{attribute 'linkalways'} 
{attribute 'no_explicit_call' := 'This FB is a CLASS and must be accessed using methods or properties'}
{attribute 'enable_dynamic_creation'}
FUNCTION_BLOCK Node_FB_VN_InitializeFunction EXTENDS VisionNode
VAR
    eFunction : _ETcVnInitializableFunction(ETcVnInitializableFunction.TCVN_IF_OCR);
    nOptions : _ULINT(0);
    bStart : _BOOL(FALSE);
    //nTimeout : 
	hresult : _HRESULT(S_OK);
END_VAR

// This is currently disabled as it's an FB and not a function.

METHOD PUBLIC  Clone : I_Node
VAR
	pNode : POINTER TO Node_FB_VN_InitializeFunction;
END_VAR
pNode := __NEW(Node_FB_VN_InitializeFunction);
Clone := pNode^;
END_METHOD

METHOD FB_init : BOOL
VAR_INPUT
	bInitRetains : BOOL; // if TRUE, the retain variables are initialized (warm start / cold start)
	bInCopyCode : BOOL;  // if TRUE, the instance afterwards gets moved into the copy code (online change)
END_VAR
AddParameter('eFunction', eFunction);
AddParameter('nOptions', nOptions);
AddParameter('bStart', bStart);
//AddParameter('nTimeout', nTimeout);
AddOutput('hresult', hresult);
END_METHOD

METHOD PROTECTED OnExecute
VAR_INST
    fbInit : FB_VN_InitializeFunction;
    fbStart : R_TRIG;
    execute : BOOL;
    result : HRESULT := -1;
END_VAR
fbStart(CLK := bStart.Value);

IF fbStart.Q AND NOT execute THEN
    execute := TRUE;
END_IF

IF execute THEN
    fbInit(eFunction := TCVN_IF_OCR, nOptions := nOptions.Value, bStart := TRUE);
    IF NOT fbInit.bBusy THEN
        fbInit(bStart := FALSE);
        IF NOT fbInit.bError THEN
            result := S_OK;
        ELSE
            result := -1;
        END_IF
        execute := FALSE;
    END_IF
END_IF

hresult.Value := result;
END_METHOD

METHOD PUBLIC PreExecutionCheck
VAR_INPUT
	Check : I_PreExecutionChecks;
END_VAR
END_METHOD

END_FUNCTION_BLOCK

(* stored: Version 1.1.0.1, ProductVersion 3.1.4026.19
   POU Node_FB_VN_InitializeFunction: Id {81dcaabb-16eb-0a21-0b7d-9e0b30687d2d}, SpecialFunc None
   Folder Constructor: Id {1d65190d-0365-048f-0e3c-580fa4c504d4}
   Method Clone: Id {fb52ccad-99d5-05b8-2a54-203e6b543320}
   Method FB_init: Id {f6f869c5-3cdc-07b1-14eb-a66c5d1ea1c0}
   Method OnExecute: Id {5600bdbe-a65e-0035-1e1d-751f798e7f4a}
   Method PreExecutionCheck: Id {db86eb7b-05a7-0790-31da-36a4ba4c9b5e} *)
